FUNCTION_BLOCK FbTriggerRS (* RS- Триггер с приоритетом на сброс. *)
  (* Standard: 61499-1; Description: Simple FB with one algorithm *)
  (* Version 2.1, 2026-03-14, VA, LIB_PLC *)
  (* Documentation:
  // RS- Триггер с приоритетом на сброс. //       DbTriggerRS //     +-------------+ //     | FbTriggerRS | //  ->-|Set       Out|->- //  ->-|Rst          | //     +-------------+  //   Релейная интерпритация.  //  |                       | //  |  Rst     Set     Out  | //  +--|/|--+--| |--+--( )--+ //  |       |       |       | //  |       |  Out  |       | //  |       +--| |--+       | //  |                       |
  *)
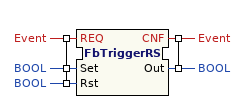
  EVENT_INPUT
    REQ WITH Set, Rst; (* Normal Execution Request *)
  END_EVENT
  EVENT_OUTPUT
    CNF WITH Out; (* Execution Confirmation *)
  END_EVENT
  VAR_INPUT
    Set : BOOL := FALSE; (* Set — установить единицу. *)
    Rst : BOOL := FALSE; (* Reset — сбросить на ноль. *)
  END_VAR
  VAR_OUTPUT
    Out : BOOL := FALSE; (* Выход триггера. *)
  END_VAR
  EC_STATES
    REQ : REQ -> CNF;
  END_STATES
  ALGORITHM REQ IN ST:
// RS- Триггер.
Out := (Out OR Set) AND (NOT (Rst));

// @COPYLEFT ALL WRONGS RESERVED :)
// Author: VA
// Contacts: DIY.PLC.314@gmail.com
// Date start LIB_PLC: 2014
// License: GNU GPL-2.0-or-later
// https://www.gnu.org/licenses/old-licenses/gpl-2.0.html
// https://www.youtube.com/watch?v=n1F_MfLRlX0
// https://www.youtube.com/@DIY_PLC
// https://github.com/DIYPLC/LIB_PLC
// https://oshwlab.com/diy.plc.314/PLC_HW1_SW1
// https://3dtoday.ru/3d-models/mechanical-parts/body/korpus-na-din-reiku
// https://t.me/DIY_PLC
  END_ALGORITHM
END_FUNCTION_BLOCK
